(* IEC 61131-3 sources: CodesysTest/alpha/export/Device.dev/Plc Logic/Application/ObjectHandling/FB_CollectionHandlerActiveFaults.pou, 2 files *)

(* ---- FB_CollectionHandlerActiveFaults.pou.st ---- *)
(*#-#-#-#-#-#-#-#-#-#---Declaration---#-#-#-#-#-#-#-#-#-#-#-#-#*)

FUNCTION_BLOCK FB_CollectionHandlerActiveFaults
VAR_INPUT
END_VAR
VAR
	Collection: ARRAY[0..GlobalObjects.MAX_FAULTS] OF IFault; // object array
	ObjNames   : ARRAY[0..GlobalObjects.MAX_FAULTS] OF STRING;
	_ArrayOver   : BOOL;
	_BadObj      : INT;
	_DupeObj   : INT;
	_OverObj   : INT;
	_TotalObj   : UINT;
END_VAR

VAR_OUTPUT
	faultActive : BOOL;
END_VAR(*#-#-#-#-#-#-#-#-#-#---Implementation---#-#-#-#-#-#-#-#-#-#-#-#-#*)

//	Function Block: FB_CollectionHandlerActiveFaults
//	Description: This collection handler adds and removes active faults to an array
//				 The add and remove methods are called from FB_Fault
//	Created by: Tom Jacobs
//	Created Date: Friday, September 7, 2018

(* ---- RemoveObject.m.st ---- *)
(*#-#-#-#-#-#-#-#-#-#---Declaration---#-#-#-#-#-#-#-#-#-#-#-#-#*)

METHOD RemoveObject
VAR_INPUT
	Obj   : IFault;
END_VAR

VAR
	I   : UINT;
	J : UINT;
END_VAR
(*#-#-#-#-#-#-#-#-#-#---Implementation---#-#-#-#-#-#-#-#-#-#-#-#-#*)

FOR I:= 0 TO _TotalObj DO
	IF Collection[I] = Obj THEN
		// object pointer matches - get rid of it
		FOR J := I TO _TotalObj DO
			Collection[J] := Collection[J+1];
			ObjNames[J]:= ObjNames[J+1];
		END_FOR
		_TotalObj := _TotalObj - 1;
		IF _TotalObj = 0 THEN
			faultActive := FALSE;
		END_IF
		RETURN;
	END_IF
END_FOR
